ORGANIZATION_BLOCK OB 100
TITLE = "Complete Restart"
VERSION : 0.1
VAR_TEMP
  OB100_EV_CLASS : BYTE ;	//16#13, Event class 1, Entering event state, Event logged in diagnostic buffer
  OB100_STRTUP : BYTE ;	//16#81/82/83/84 Method of startup
  OB100_PRIORITY : BYTE ;	//27 (Priority of 1 is lowest)
  OB100_OB_NUMBR : BYTE ;	//100 (Organization block 100, OB100)
  OB100_RESERVED_1 : BYTE ;	//Reserved for system
  OB100_RESERVED_2 : BYTE ;	//Reserved for system
  OB100_STOP : WORD ;	//Event that caused CPU to stop (16#4xxx)
  OB100_STRT_INFO : DWORD ;	//Information on how system started
  OB100_DATE_TIME : DATE_AND_TIME ;	//Date and time OB100 started
END_VAR
BEGIN
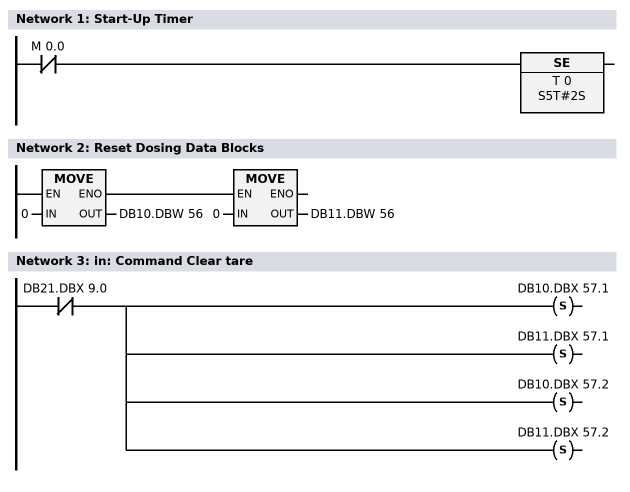
NETWORK
TITLE = Start-Up Timer
      AN    M 0.0;
      L     S5T#2S;
      SE    T 0;
NETWORK
TITLE = Reset Dosing Data Blocks
      A(;
      L     0;
      T     DB10.DBW 56;
      SET;
      SAVE;
      CLR;
      A     BR;
      );
      JNB   _001;
      L     0;
      T     DB11.DBW 56;
_001: NOP   0;
NETWORK
TITLE = in: Command Clear tare
      AN    DB21.DBX 9.0;
      S     DB10.DBX 57.1;
      S     DB11.DBX 57.1;
      S     DB10.DBX 57.2;
      S     DB11.DBX 57.2;
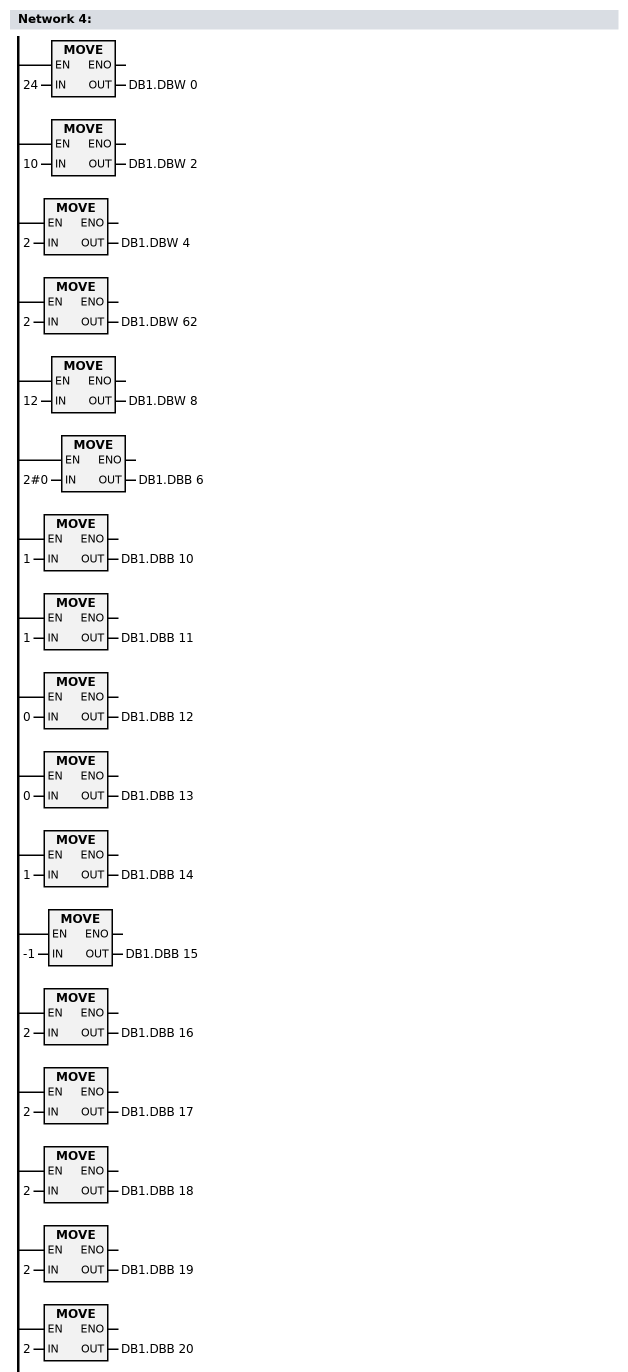
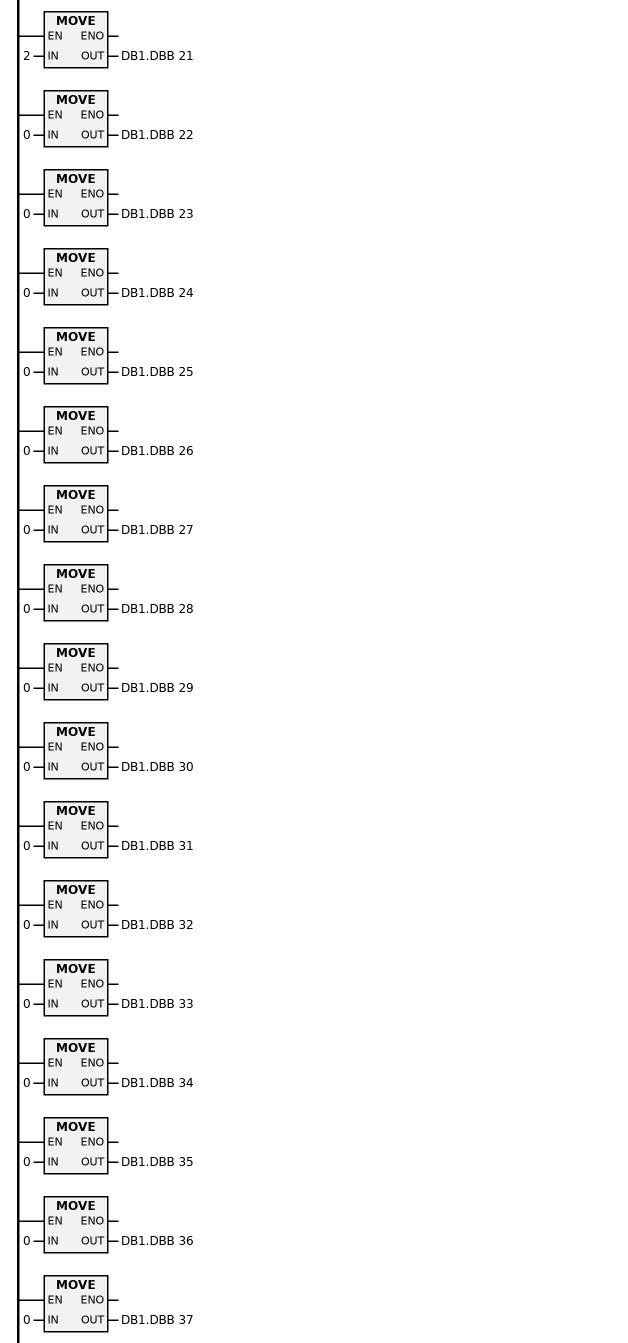
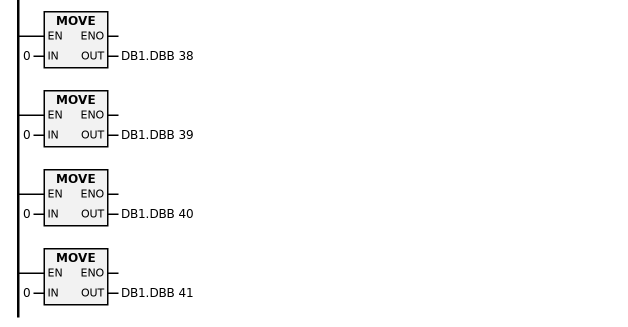
NETWORK
TITLE =
      L     24;
      T     DB1.DBW 0;
      L     10;
      T     DB1.DBW 2;
      L     2;
      T     DB1.DBW 4;
      L     2;
      T     DB1.DBW 62;
      L     12;
      T     DB1.DBW 8;
      L     2#0;
      T     DB1.DBB 6;
// 1: main scale
// 2: sub scale
// 3: color scale
      L     1;
      T     DB1.DBB 10;
      L     1;
      T     DB1.DBB 11;
      L     0;
      T     DB1.DBB 12;
      L     0;
      T     DB1.DBB 13;
      L     1;
      T     DB1.DBB 14;
      L     -1;
      T     DB1.DBB 15;
      L     2;
      T     DB1.DBB 16;
      L     2;
      T     DB1.DBB 17;
      L     2;
      T     DB1.DBB 18;
      L     2;
      T     DB1.DBB 19;
      L     2;
      T     DB1.DBB 20;
      L     2;
      T     DB1.DBB 21;
      L     0;
      T     DB1.DBB 22;
      L     0;
      T     DB1.DBB 23;
      L     0;
      T     DB1.DBB 24;
      L     0;
      T     DB1.DBB 25;
      L     0;
      T     DB1.DBB 26;
      L     0;
      T     DB1.DBB 27;
      L     0;
      T     DB1.DBB 28;
      L     0;
      T     DB1.DBB 29;
      L     0;
      T     DB1.DBB 30;
      L     0;
      T     DB1.DBB 31;
      L     0;
      T     DB1.DBB 32;
      L     0;
      T     DB1.DBB 33;
      L     0;
      T     DB1.DBB 34;
      L     0;
      T     DB1.DBB 35;
      L     0;
      T     DB1.DBB 36;
      L     0;
      T     DB1.DBB 37;
      L     0;
      T     DB1.DBB 38;
      L     0;
      T     DB1.DBB 39;
      L     0;
      T     DB1.DBB 40;
      L     0;
      T     DB1.DBB 41;
NETWORK
TITLE = init CP Gravimet
      L     160;
      T     DB1.DBW 64;
      L     10;
      T     DB1.DBW 66;
      L     DB23.DBW 34;
      L     DB1.DBW 64;
      <I;
      JC    err1;
      L     DB1.DBW 64;
      L     DB1.DBW 66;
      +I;
      L     DB23.DBW 34;
      TAK;
      >=I;
      JC    err1;
      JU    go1;
err1: L     DB1.DBW 64;
      T     DB23.DBW 34;
go1:  NOP   0;
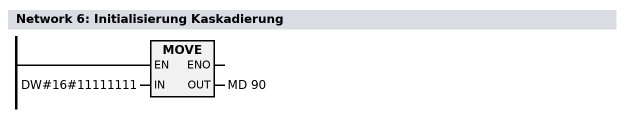
NETWORK
TITLE = Initialisierung Kaskadierung
      L     DW#16#11111111;
      T     MD 90;
END_ORGANIZATION_BLOCK

ORGANIZATION_BLOCK OB 121
TITLE = "Programming Error"
VERSION : 0.1
VAR_TEMP
  OB121_EV_CLASS : BYTE ;	//16#25, Event class 2, Entering event state, Internal fault event
  OB121_SW_FLT : BYTE ;	//16#XX Software programming fault
  OB121_PRIORITY : BYTE ;	//Priority of OB Execution
  OB121_OB_NUMBR : BYTE ;	//121 (Organization block 121, OB121)
  OB121_BLK_TYPE : BYTE ;	//16#88/8A/8B/8C/8E Type of block fault occured in
  OB121_RESERVED_1 : BYTE ;	//Reserved for system
  OB121_FLT_REG : WORD ;	//16#XX Specific register that caused fault
  OB121_BLK_NUM : WORD ;	//Number of block that programming fault occured in
  OB121_PRG_ADDR : WORD ;	//Address in block where programming fault occured
  OB121_DATE_TIME : DATE_AND_TIME ;	//Date and time OB121 started
END_VAR
BEGIN
// (block stored without names or comments; labels and parameter names are numbered)
END_ORGANIZATION_BLOCK

ORGANIZATION_BLOCK OB 122
TITLE = "Module Access Error"
VERSION : 0.1
VAR_TEMP
  OB122_EV_CLASS : BYTE ;	//16#29, Event class 2, Entering event state, Internal fault event
  OB122_SW_FLT : BYTE ;	//16#XX Software error code
  OB122_PRIORITY : BYTE ;	//Priority of OB Execution
  OB122_OB_NUMBR : BYTE ;	//122 (Organization block 122, OB122)
  OB122_BLK_TYPE : BYTE ;	//16#88/8C/8E Type of block fault occured in
  OB122_MEM_AREA : BYTE ;	//Memory area where access error occured
  OB122_MEM_ADDR : WORD ;	//Memory address where access error occured
  OB122_BLK_NUM : WORD ;	//Block number in which error occured
  OB122_PRG_ADDR : WORD ;	//Program address where error occured
  OB122_DATE_TIME : DATE_AND_TIME ;	//Date and time OB1 started
END_VAR
BEGIN
// (block stored without names or comments; labels and parameter names are numbered)
END_ORGANIZATION_BLOCK
